(*
  This fb is the master controller of modules.
  Like an interface handler/provider for Module to Main communiation
*)
FUNCTION_BLOCK FB_ModuleMaster EXTENDS T_NamedBase IMPLEMENTS I_ModuleMaster, I_HardwarePool
VAR
  // references
  _pPU : POINTER TO FB_PU;
  _iHwPool : I_HardwarePool;
  
  _pMasterModule : POINTER TO FB_PrintModule_Base;
END_VAR



// Noting to do

PROPERTY iHardwarePool : I_HardwarePool
GET
iHardwarePool := _iHwPool;
END_GET
END_PROPERTY

PROPERTY iMasterPrintPosition : I_PrintPosition
GET
IF _pMasterModule = 0 THEN RETURN; END_IF

iMasterPrintPosition := _pMasterModule^.iPrintPosition;
END_GET
END_PROPERTY

METHOD Init : BOOL
VAR_INPUT
  pPU : POINTER TO FB_PU;
  iHwPool : I_HardwarePool;
END_VAR
IF pPU = 0 OR iHwPool = 0 THEN LogError('init() invalid init parameter'); RETURN; END_IF

_pPU := pPU;
_iHwPool := iHwPool;
END_METHOD

METHOD registerPc : BOOL
VAR_INPUT
	pNewPc	: POINTER TO CalmarCompPrint.FB_PC;
END_VAR
_iHwPool.registerPc(pNewPc:=pNewPc);
END_METHOD

METHOD registerPh : BOOL
VAR_INPUT
	pNewPh	: POINTER TO CalmarCompPrint.FB_PH;
END_VAR
_iHwPool.registerPh(pNewPh:=pNewPh);
END_METHOD

(*
  Register for PU StatusClient
*)
METHOD registerPuStatusClient : BOOL
VAR_INPUT
	sClient	: CalmarCompPrint.I_PrintStatusClient;
END_VAR
registerPuStatusClient := _pPU^.registerStatusClient(sClient:=sClient);
END_METHOD

METHOD registerPuSubystem : BOOL
VAR_INPUT
	iSubSys	: I_PrintSubsystem;
END_VAR
_pPU^.registerStatusClient(sClient := iSubSys);
_pPU^.registerSubystem(sSubSys:= iSubSys);
END_METHOD

METHOD setMasterModule : BOOL
VAR_INPUT
  pModule : POINTER TO FB_PrintModule_Base;
END_VAR
// note make this a private method if MasterModule knows it modules
IF pModule = 0 THEN LogError('setMasterModule: invalid module given, ignore'); RETURN; END_IF

_pMasterModule := pModule;
END_METHOD

END_FUNCTION_BLOCK

(* stored: Version 1.1.0.1, ProductVersion 3.1.4024.11
   POU FB_ModuleMaster: Id {d174fcea-8a30-4fbf-8484-3c054af3ade2}, SpecialFunc None
   Folder I_HardwarePool: Id {f7cf7209-17a6-41b9-9db7-2cb856085d44}
   Folder I_ModuleMaster: Id {96598412-2f6b-42bc-90f9-92e56d561add}
   Property iHardwarePool: Id {a847ca78-a2f3-4e9b-8e9d-71d00c55cae8}
   Get Get: Id {d9d0d816-0eab-497b-aa8b-b6c3586e2191}
   Property iMasterPrintPosition: Id {df366969-a76e-4b45-acd7-0d54f39708ef}
   Get Get: Id {986a3c62-960e-4fbd-adda-e849e845e901}
   Method Init: Id {9211467c-5c9b-41c8-a36e-23ed4e2b55b2}
   Method registerPc: Id {5d9de9ad-1299-41df-bd83-47f2b3d4a0f4}
   Method registerPh: Id {0f191415-4cf5-4595-8669-cd2ca33f11d7}
   Method registerPuStatusClient: Id {e2476ae7-981b-4329-bb18-d3f85fad3146}
   Method registerPuSubystem: Id {359e2db7-fa5d-424c-bc4d-0ea6eff60e9a}
   Method setMasterModule: Id {e2704455-e4dc-4ab4-9587-790388a55ee0} *)
